(* IEC 61131-3 sources: eCockpitGit/test_project/src/%F%02 System/%F%03 LoadSaveManager/%POU%FB_LoadSave/%F%Save/%F%Structure, 5 files *)

(* ---- %METH%addKey.st ---- *)
//This adds a key and a value to the buffer
// |**Version**|**Author**| **Date** |**Changes**
// | 1         | NSN      | 22-06-20 | Creation
METHOD addKey : BOOL
VAR_INPUT
	name			:POINTER TO EASCII;	//Address of string for the tag name text
END_VAR
(*%!%__DELIMITER__%!%*)
addKey			:=		writer.addKey(name:=name);
IF doLogInt THEN
	keyFound	:=		reader.findKey(name:=name) <> EStructType.none;
END_IF

(* ---- %METH%arrayStart.st ---- *)
//This starts a new array
// |**Version**|**Author**| **Date** |**Changes**
// | 1         | NSN      | 22-06-20 | Creation
METHOD arrayStart : BOOL
VAR_INPUT
	singleLine		:BOOL;
END_VAR
(*%!%__DELIMITER__%!%*)
arrayStart		:=		writer.arrayStart(singleLine:=singleLine);
IF doLogInt THEN
	IF selectedType = EStructType.tArray THEN
		reader.nextArray();
	END_IF
	IF NOT(reader.enterObjectArray()) THEN
		logCorrection		:=		logCorrection + 1;
	END_IF
END_IF

(* ---- %METH%objectStart.st ---- *)
//This starts a new object
// |**Version**|**Author**| **Date** |**Changes**
// | 1         | NSN      | 22-06-20 | Creation
METHOD objectStart : BOOL
VAR_INPUT
	singleLine		:BOOL;
END_VAR
(*%!%__DELIMITER__%!%*)
objectStart		:=		writer.objectStart(singleLine:=singleLine);
IF doLogInt THEN
	IF selectedType = EStructType.tArray THEN
		reader.nextArray();
	END_IF
	IF NOT(reader.enterObjectArray()) THEN
		logCorrection		:=		logCorrection + 1;
	END_IF
END_IF

(* ---- %METH%structEnd.st ---- *)
//This ends the previously started object
// |**Version**|**Author**| **Date** |**Changes**
// | 1         | NSN      | 22-06-20 | Creation
METHOD structEnd : BOOL

(*%!%__DELIMITER__%!%*)
structEnd		:=		writer.structEnd();
IF doLogInt THEN
	IF logCorrection > 0 THEN
		logCorrection		:=		logCorrection - 1;
	ELSE
		reader.exitObjectArray();
	END_IF
END_IF

(* ---- %PRO%maxSize.st ---- *)
{"external": false, "compiler_defines": "", "link_always": false, "exclude_from_build": false, "enable_system_call": false}
PROPERTY maxSize : DWORD
!__GETTER__!
//This gets the amount of bytes in the buffer
// | 1         | NSN      | 22-06-20 | Creation
VAR
END_VAR

!__IMPLEMENTATION__!
maxSize		:=		writer.maxSize;
!__SETTER__!
